TYPE Motor_Error :
(   
	NO_ERROR,
	START_TIMEOUT,
	FEEDBACK_LOST,
	INTERLOCKM_OPEN,
	ESTOP_ACTIVE
);
END_TYPE

(* stored: Version 1.1.0.1, ProductVersion 3.1.4024.16
   DUT Motor_Error: Id {d3996b44-0d43-4097-8a21-82a25477c9fc} *)
